{attribute 'qualified_only'}
{attribute 'strict'}
TYPE GearRole :
(
  Undefined
	,Primary
  ,SecondarySimple
  ,SecondaryStruckig
);
END_TYPE

(* stored: Version 1.1.0.1
   DUT GearRole: Id {002975d2-f5bb-4381-ad3b-3b7683ea35e1} *)
